REGION Network 20
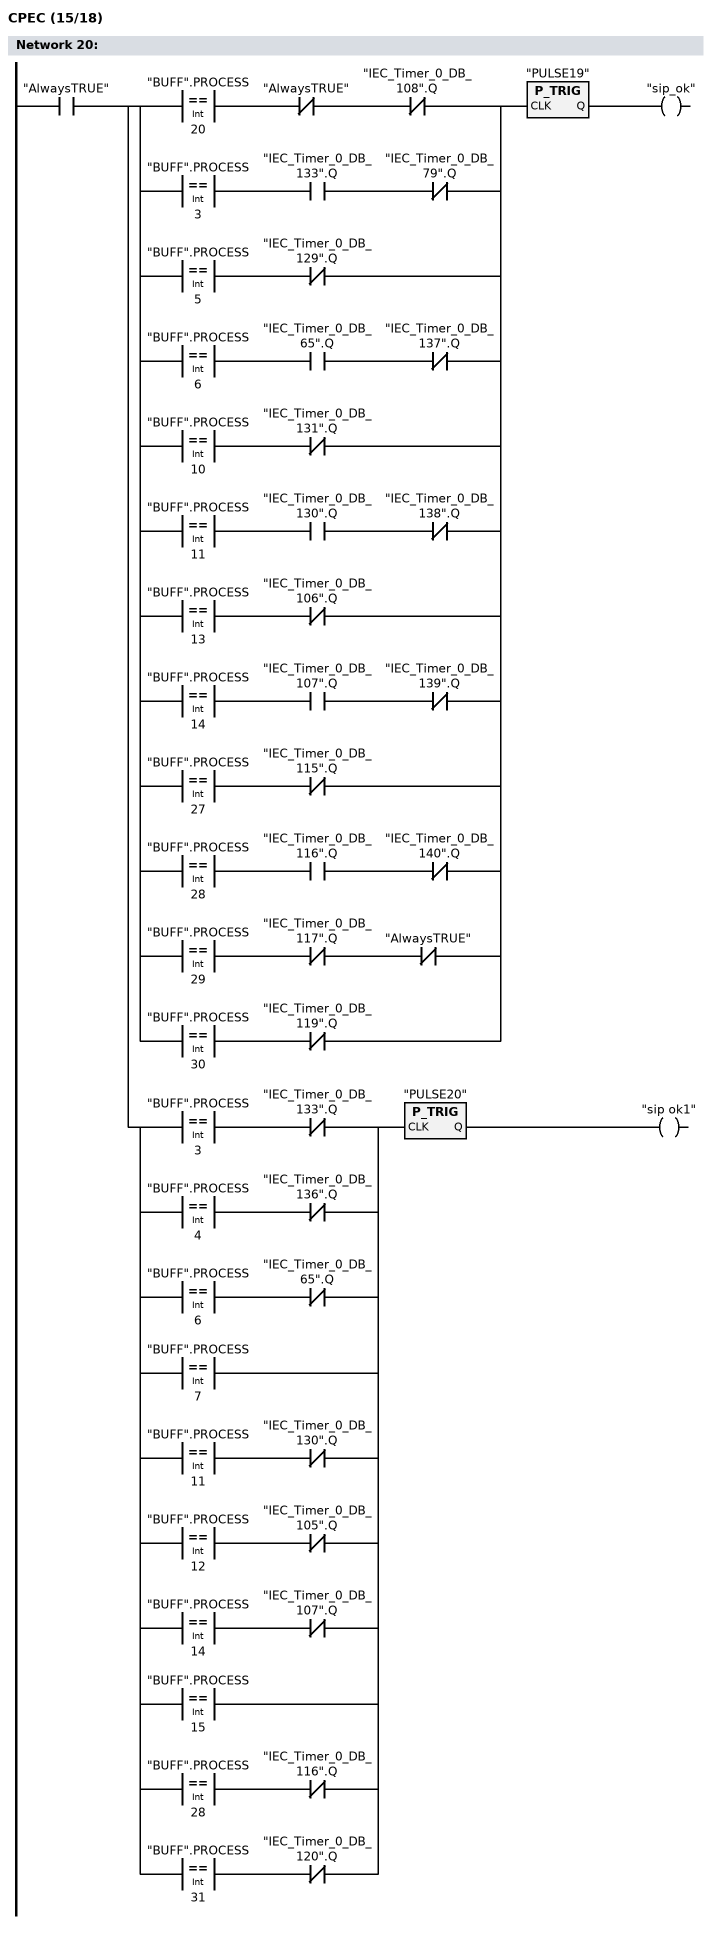
   RUNG wire#powerrail
      Contact( "AlwaysTRUE" )
      wire#w1
      { S7_Templates := "SrcType := Int" } EQ_Contact(in1 := "BUFF".PROCESS, in2 := 20)
      I_Contact( "AlwaysTRUE" )
      I_Contact( "IEC_Timer_0_DB_108".Q )
      wire#w2
      P_Trig( "PULSE19" )
      Coil( "sip_ok" )
   END_RUNG
   RUNG wire#w1
      { S7_Templates := "SrcType := Int" } EQ_Contact(in1 := "BUFF".PROCESS, in2 := 3)
      Contact( "IEC_Timer_0_DB_133".Q )
      I_Contact( "IEC_Timer_0_DB_79".Q )
   END_RUNG wire#w2
   RUNG wire#w1
      { S7_Templates := "SrcType := Int" } EQ_Contact(in1 := "BUFF".PROCESS, in2 := 5)
      I_Contact( "IEC_Timer_0_DB_129".Q )
   END_RUNG wire#w2
   RUNG wire#w1
      { S7_Templates := "SrcType := Int" } EQ_Contact(in1 := "BUFF".PROCESS, in2 := 6)
      Contact( "IEC_Timer_0_DB_65".Q )
      I_Contact( "IEC_Timer_0_DB_137".Q )
   END_RUNG wire#w2
   RUNG wire#w1
      { S7_Templates := "SrcType := Int" } EQ_Contact(in1 := "BUFF".PROCESS, in2 := 10)
      I_Contact( "IEC_Timer_0_DB_131".Q )
   END_RUNG wire#w2
   RUNG wire#w1
      { S7_Templates := "SrcType := Int" } EQ_Contact(in1 := "BUFF".PROCESS, in2 := 11)
      Contact( "IEC_Timer_0_DB_130".Q )
      I_Contact( "IEC_Timer_0_DB_138".Q )
   END_RUNG wire#w2
   RUNG wire#w1
      { S7_Templates := "SrcType := Int" } EQ_Contact(in1 := "BUFF".PROCESS, in2 := 13)
      I_Contact( "IEC_Timer_0_DB_106".Q )
   END_RUNG wire#w2
   RUNG wire#w1
      { S7_Templates := "SrcType := Int" } EQ_Contact(in1 := "BUFF".PROCESS, in2 := 14)
      Contact( "IEC_Timer_0_DB_107".Q )
      I_Contact( "IEC_Timer_0_DB_139".Q )
   END_RUNG wire#w2
   RUNG wire#w1
      { S7_Templates := "SrcType := Int" } EQ_Contact(in1 := "BUFF".PROCESS, in2 := 27)
      I_Contact( "IEC_Timer_0_DB_115".Q )
   END_RUNG wire#w2
   RUNG wire#w1
      { S7_Templates := "SrcType := Int" } EQ_Contact(in1 := "BUFF".PROCESS, in2 := 28)
      Contact( "IEC_Timer_0_DB_116".Q )
      I_Contact( "IEC_Timer_0_DB_140".Q )
   END_RUNG wire#w2
   RUNG wire#w1
      { S7_Templates := "SrcType := Int" } EQ_Contact(in1 := "BUFF".PROCESS, in2 := 29)
      I_Contact( "IEC_Timer_0_DB_117".Q )
      I_Contact( "AlwaysTRUE" )
   END_RUNG wire#w2
   RUNG wire#w1
      { S7_Templates := "SrcType := Int" } EQ_Contact(in1 := "BUFF".PROCESS, in2 := 30)
      I_Contact( "IEC_Timer_0_DB_119".Q )
   END_RUNG wire#w2
   RUNG wire#w1
      { S7_Templates := "SrcType := Int" } EQ_Contact(in1 := "BUFF".PROCESS, in2 := 3)
      I_Contact( "IEC_Timer_0_DB_133".Q )
      wire#w3
      P_Trig( "PULSE20" )
      Coil( "sip ok1" )
   END_RUNG
   RUNG wire#w1
      { S7_Templates := "SrcType := Int" } EQ_Contact(in1 := "BUFF".PROCESS, in2 := 4)
      I_Contact( "IEC_Timer_0_DB_136".Q )
   END_RUNG wire#w3
   RUNG wire#w1
      { S7_Templates := "SrcType := Int" } EQ_Contact(in1 := "BUFF".PROCESS, in2 := 6)
      I_Contact( "IEC_Timer_0_DB_65".Q )
   END_RUNG wire#w3
   RUNG wire#w1
      { S7_Templates := "SrcType := Int" } EQ_Contact(in1 := "BUFF".PROCESS, in2 := 7)
   END_RUNG wire#w3
   RUNG wire#w1
      { S7_Templates := "SrcType := Int" } EQ_Contact(in1 := "BUFF".PROCESS, in2 := 11)
      I_Contact( "IEC_Timer_0_DB_130".Q )
   END_RUNG wire#w3
   RUNG wire#w1
      { S7_Templates := "SrcType := Int" } EQ_Contact(in1 := "BUFF".PROCESS, in2 := 12)
      I_Contact( "IEC_Timer_0_DB_105".Q )
   END_RUNG wire#w3
   RUNG wire#w1
      { S7_Templates := "SrcType := Int" } EQ_Contact(in1 := "BUFF".PROCESS, in2 := 14)
      I_Contact( "IEC_Timer_0_DB_107".Q )
   END_RUNG wire#w3
   RUNG wire#w1
      { S7_Templates := "SrcType := Int" } EQ_Contact(in1 := "BUFF".PROCESS, in2 := 15)
   END_RUNG wire#w3
   RUNG wire#w1
      { S7_Templates := "SrcType := Int" } EQ_Contact(in1 := "BUFF".PROCESS, in2 := 28)
      I_Contact( "IEC_Timer_0_DB_116".Q )
   END_RUNG wire#w3
   RUNG wire#w1
      { S7_Templates := "SrcType := Int" } EQ_Contact(in1 := "BUFF".PROCESS, in2 := 31)
      I_Contact( "IEC_Timer_0_DB_120".Q )
   END_RUNG wire#w3
   // the same network as SCL:
   #_w1 := "AlwaysTRUE" AND ((("BUFF".PROCESS = 20) AND NOT "AlwaysTRUE" AND NOT "IEC_Timer_0_DB_108".Q) OR (("BUFF".PROCESS = 3) AND "IEC_Timer_0_DB_133".Q AND NOT "IEC_Timer_0_DB_79".Q) OR (("BUFF".PROCESS = 5) AND NOT "IEC_Timer_0_DB_129".Q) OR (("BUFF".PROCESS = 6) AND "IEC_Timer_0_DB_65".Q AND NOT "IEC_Timer_0_DB_137".Q) OR (("BUFF".PROCESS = 10) AND NOT "IEC_Timer_0_DB_131".Q) OR (("BUFF".PROCESS = 11) AND "IEC_Timer_0_DB_130".Q AND NOT "IEC_Timer_0_DB_138".Q) OR (("BUFF".PROCESS = 13) AND NOT "IEC_Timer_0_DB_106".Q) OR (("BUFF".PROCESS = 14) AND "IEC_Timer_0_DB_107".Q AND NOT "IEC_Timer_0_DB_139".Q) OR (("BUFF".PROCESS = 27) AND NOT "IEC_Timer_0_DB_115".Q) OR (("BUFF".PROCESS = 28) AND "IEC_Timer_0_DB_116".Q AND NOT "IEC_Timer_0_DB_140".Q) OR (("BUFF".PROCESS = 29) AND NOT "IEC_Timer_0_DB_117".Q AND NOT "AlwaysTRUE") OR (("BUFF".PROCESS = 30) AND NOT "IEC_Timer_0_DB_119".Q));
   #_w2 := #_w1 AND NOT "PULSE19";   // rising edge
   "PULSE19" := #_w1;
   "sip_ok" := #_w2;
   #_w3 := "AlwaysTRUE" AND ((("BUFF".PROCESS = 3) AND NOT "IEC_Timer_0_DB_133".Q) OR (("BUFF".PROCESS = 4) AND NOT "IEC_Timer_0_DB_136".Q) OR (("BUFF".PROCESS = 6) AND NOT "IEC_Timer_0_DB_65".Q) OR ("BUFF".PROCESS = 7) OR (("BUFF".PROCESS = 11) AND NOT "IEC_Timer_0_DB_130".Q) OR (("BUFF".PROCESS = 12) AND NOT "IEC_Timer_0_DB_105".Q) OR (("BUFF".PROCESS = 14) AND NOT "IEC_Timer_0_DB_107".Q) OR ("BUFF".PROCESS = 15) OR (("BUFF".PROCESS = 28) AND NOT "IEC_Timer_0_DB_116".Q) OR (("BUFF".PROCESS = 31) AND NOT "IEC_Timer_0_DB_120".Q));
   #_w4 := #_w3 AND NOT "PULSE20";   // rising edge
   "PULSE20" := #_w3;
   "sip ok1" := #_w4;
END_REGION

REGION Network 21
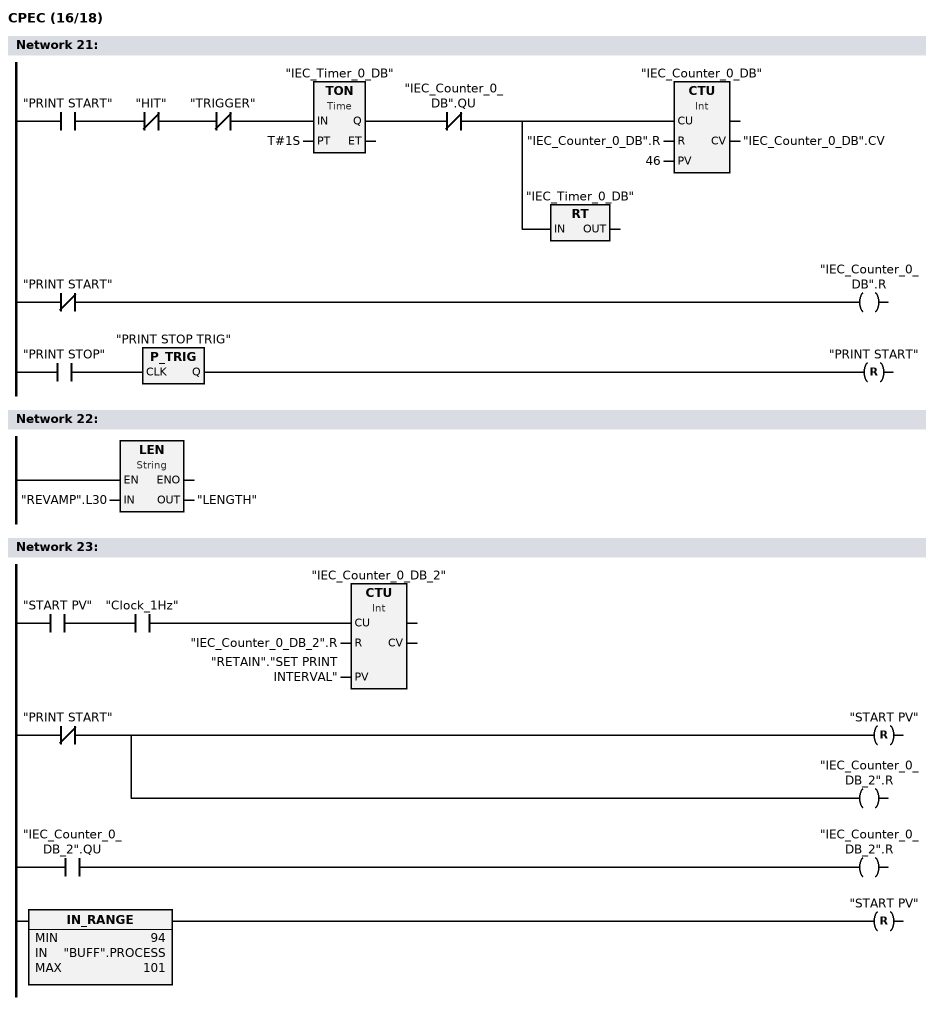
   RUNG wire#powerrail
      Contact( "PRINT START" )
      I_Contact( "HIT" )
      I_Contact( "TRIGGER" )
      { S7_Templates := "time_type := Time" } "IEC_Timer_0_DB".TON(pt := T#1S, et =>)
      I_Contact( "IEC_Counter_0_DB".QU )
      wire#w1
      { S7_Templates := "value_type := Int" } "IEC_Counter_0_DB".CTU(r := "IEC_Counter_0_DB".R, pv := 46, cv => "IEC_Counter_0_DB".CV)
   END_RUNG
   RUNG wire#w1
      RT_Coil( "IEC_Timer_0_DB" )
   END_RUNG
   RUNG wire#powerrail
      I_Contact( "PRINT START" )
      Coil( "IEC_Counter_0_DB".R )
   END_RUNG
   RUNG wire#powerrail
      Contact( "PRINT STOP" )
      P_Trig( "PRINT STOP TRIG" )
      R_Coil( "PRINT START" )
   END_RUNG
   // the same network as SCL:
   "IEC_Timer_0_DB".TON(IN := "PRINT START" AND NOT "HIT" AND NOT "TRIGGER", PT := T#1S);
   #_w1 := "IEC_Timer_0_DB".Q AND NOT "IEC_Counter_0_DB".QU;
   "IEC_Counter_0_DB".CTU(CU := #_w1, R := "IEC_Counter_0_DB".R, PV := 46, CV => "IEC_Counter_0_DB".CV);
   IF #_w1 THEN RESET_TIMER("IEC_Timer_0_DB"); END_IF;
   "IEC_Counter_0_DB".R := NOT "PRINT START";
   #_w2 := "PRINT STOP" AND NOT "PRINT STOP TRIG";   // rising edge
   "PRINT STOP TRIG" := "PRINT STOP";
   IF #_w2 THEN "PRINT START" := FALSE; END_IF;
END_REGION

REGION Network 22
   RUNG wire#powerrail
      { S7_Templates := "[str_type := String, return_type := Int]" } LEN(IN := "REVAMP".L30, OUT => "LENGTH")
   END_RUNG
   // the same network as SCL:
   LEN(IN := "REVAMP".L30, OUT => "LENGTH");
END_REGION

REGION Network 23
   RUNG wire#powerrail
      Contact( "START PV" )
      Contact( "Clock_1Hz" )
      { S7_Templates := "value_type := Int" } "IEC_Counter_0_DB_2".CTU(r := "IEC_Counter_0_DB_2".R, pv := "RETAIN"."SET PRINT INTERVAL", cv =>)
   END_RUNG
   RUNG wire#powerrail
      I_Contact( "PRINT START" )
      wire#w1
      R_Coil( "START PV" )
   END_RUNG
   RUNG wire#w1
      Coil( "IEC_Counter_0_DB_2".R )
   END_RUNG
   RUNG wire#powerrail
      Contact( "IEC_Counter_0_DB_2".QU )
      Coil( "IEC_Counter_0_DB_2".R )
   END_RUNG
   RUNG wire#powerrail
      { S7_Templates := "SrcType := Int" } InRange(min := 94, in := "BUFF".PROCESS, max := 101)
      R_Coil( "START PV" )
   END_RUNG
   // the same network as SCL:
   "IEC_Counter_0_DB_2".CTU(CU := "START PV" AND "Clock_1Hz",
                           R := "IEC_Counter_0_DB_2".R,
                           PV := "RETAIN"."SET PRINT INTERVAL");
   IF NOT "PRINT START" THEN "START PV" := FALSE; END_IF;
   "IEC_Counter_0_DB_2".R := NOT "PRINT START";
   "IEC_Counter_0_DB_2".R := "IEC_Counter_0_DB_2".QU;
   IF (94 <= "BUFF".PROCESS) AND ("BUFF".PROCESS <= 101) THEN "START PV" := FALSE; END_IF;
END_REGION

REGION Network 24
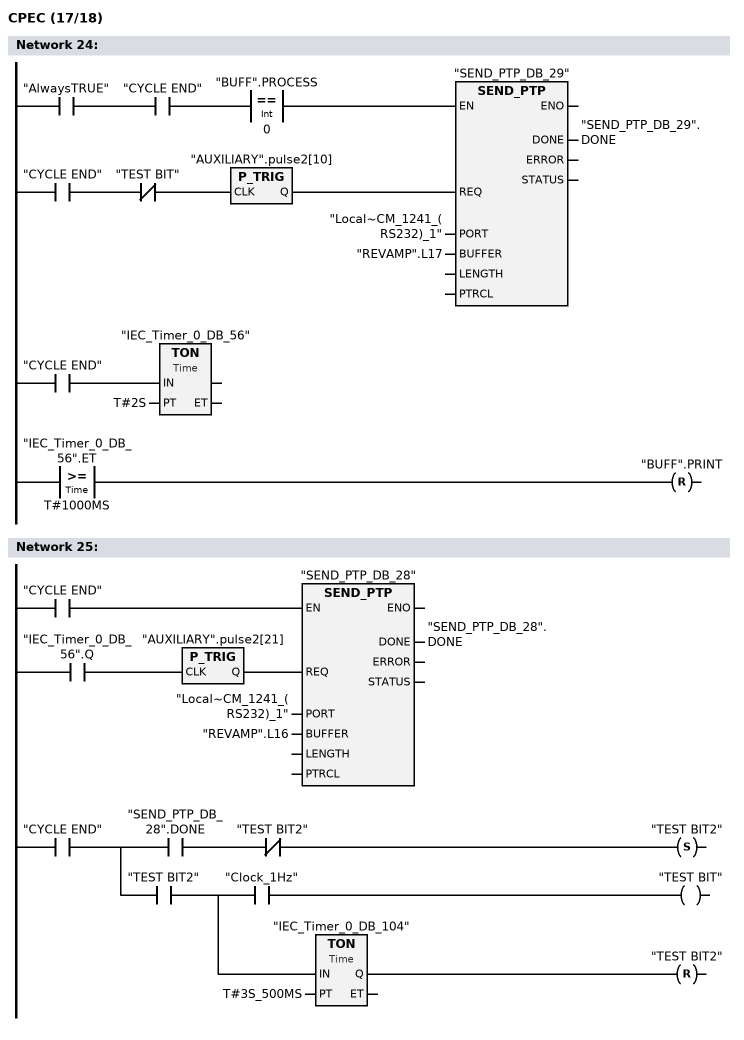
   RUNG wire#powerrail
      Contact( "AlwaysTRUE" )
      Contact( "CYCLE END" )
      { S7_Templates := "SrcType := Int" } EQ_Contact(in1 := "BUFF".PROCESS, in2 := 0)
      "SEND_PTP_DB_29".SEND_PTP(REQ := wire#w1, PORT := "Local~CM_1241_(RS232)_1", BUFFER := "REVAMP".L17, LENGTH :=, PTRCL :=, DONE => "SEND_PTP_DB_29".DONE, ERROR =>, STATUS =>)
   END_RUNG
   RUNG wire#powerrail
      Contact( "CYCLE END" )
      I_Contact( "TEST BIT" )
      P_Trig( "AUXILIARY".pulse2[10] )
   END_RUNG wire#w1
   RUNG wire#powerrail
      Contact( "CYCLE END" )
      { S7_Templates := "time_type := Time" } "IEC_Timer_0_DB_56".TON(pt := T#2S, et =>)
   END_RUNG
   RUNG wire#powerrail
      { S7_Templates := "SrcType := Time" } GE_Contact(in1 := "IEC_Timer_0_DB_56".ET, in2 := T#1000MS)
      R_Coil( "BUFF".PRINT )
   END_RUNG
   // the same network as SCL:
   #_w1 := "CYCLE END" AND NOT "TEST BIT";
   #_w2 := #_w1 AND NOT "AUXILIARY".pulse2[10];   // rising edge
   "AUXILIARY".pulse2[10] := #_w1;
   IF "AlwaysTRUE" AND "CYCLE END" AND ("BUFF".PROCESS = 0) THEN
       "SEND_PTP_DB_29"(REQ := #_w2,   // SEND_PTP
                        PORT := "Local~CM_1241_(RS232)_1",
                        BUFFER := "REVAMP".L17,
                        DONE => "SEND_PTP_DB_29".DONE);
   END_IF;
   "IEC_Timer_0_DB_56".TON(IN := "CYCLE END", PT := T#2S);
   IF "IEC_Timer_0_DB_56".ET >= T#1000MS THEN "BUFF".PRINT := FALSE; END_IF;
END_REGION

REGION Network 25
   RUNG wire#powerrail
      Contact( "CYCLE END" )
      "SEND_PTP_DB_28".SEND_PTP(REQ := wire#w1, PORT := "Local~CM_1241_(RS232)_1", BUFFER := "REVAMP".L16, LENGTH :=, PTRCL :=, DONE => "SEND_PTP_DB_28".DONE, ERROR =>, STATUS =>)
   END_RUNG
   RUNG wire#powerrail
      Contact( "IEC_Timer_0_DB_56".Q )
      P_Trig( "AUXILIARY".pulse2[21] )
   END_RUNG wire#w1
   RUNG wire#powerrail
      Contact( "CYCLE END" )
      wire#w2
      Contact( "SEND_PTP_DB_28".DONE )
      I_Contact( "TEST BIT2" )
      S_Coil( "TEST BIT2" )
   END_RUNG
   RUNG wire#w2
      Contact( "TEST BIT2" )
      wire#w3
      Contact( "Clock_1Hz" )
      Coil( "TEST BIT" )
   END_RUNG
   RUNG wire#w3
      { S7_Templates := "time_type := Time" } "IEC_Timer_0_DB_104".TON(pt := T#3S_500MS, et =>)
      R_Coil( "TEST BIT2" )
   END_RUNG
   // the same network as SCL:
   #_w1 := "IEC_Timer_0_DB_56".Q AND NOT "AUXILIARY".pulse2[21];   // rising edge
   "AUXILIARY".pulse2[21] := "IEC_Timer_0_DB_56".Q;
   IF "CYCLE END" THEN
       "SEND_PTP_DB_28"(REQ := #_w1,   // SEND_PTP
                        PORT := "Local~CM_1241_(RS232)_1",
                        BUFFER := "REVAMP".L16,
                        DONE => "SEND_PTP_DB_28".DONE);
   END_IF;
   IF "CYCLE END" AND "SEND_PTP_DB_28".DONE AND NOT "TEST BIT2" THEN "TEST BIT2" := TRUE; END_IF;
   #_w2 := "CYCLE END" AND "TEST BIT2";
   "TEST BIT" := #_w2 AND "Clock_1Hz";
   "IEC_Timer_0_DB_104".TON(IN := #_w2, PT := T#3S_500MS);
   IF "IEC_Timer_0_DB_104".Q THEN "TEST BIT2" := FALSE; END_IF;
END_REGION

REGION Network 26
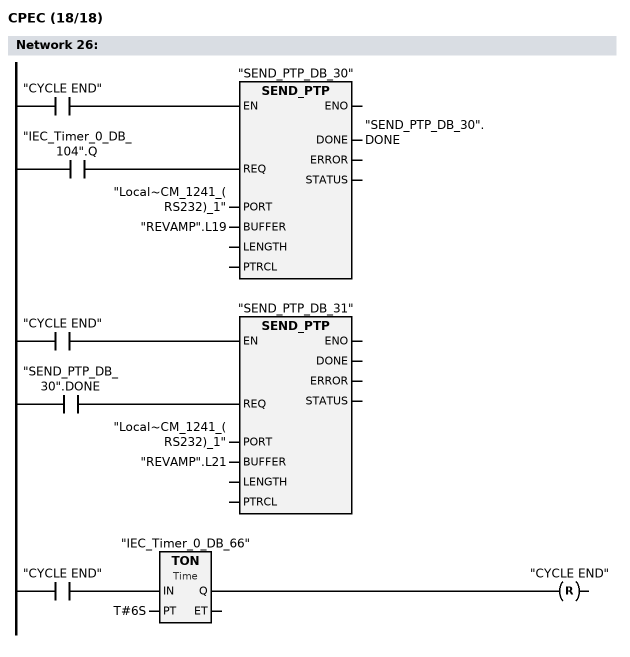
   RUNG wire#powerrail
      Contact( "CYCLE END" )
      "SEND_PTP_DB_30".SEND_PTP(REQ := wire#w1, PORT := "Local~CM_1241_(RS232)_1", BUFFER := "REVAMP".L19, LENGTH :=, PTRCL :=, DONE => "SEND_PTP_DB_30".DONE, ERROR =>, STATUS =>)
   END_RUNG
   RUNG wire#powerrail
      Contact( "IEC_Timer_0_DB_104".Q )
   END_RUNG wire#w1
   RUNG wire#powerrail
      Contact( "CYCLE END" )
      "SEND_PTP_DB_31".SEND_PTP(REQ := wire#w2, PORT := "Local~CM_1241_(RS232)_1", BUFFER := "REVAMP".L21, LENGTH :=, PTRCL :=, DONE =>, ERROR =>, STATUS =>)
   END_RUNG
   RUNG wire#powerrail
      Contact( "SEND_PTP_DB_30".DONE )
   END_RUNG wire#w2
   RUNG wire#powerrail
      Contact( "CYCLE END" )
      { S7_Templates := "time_type := Time" } "IEC_Timer_0_DB_66".TON(pt := T#6S, et =>)
      R_Coil( "CYCLE END" )
   END_RUNG
   // the same network as SCL:
   IF "CYCLE END" THEN
       "SEND_PTP_DB_30"(REQ := "IEC_Timer_0_DB_104".Q,   // SEND_PTP
                        PORT := "Local~CM_1241_(RS232)_1",
                        BUFFER := "REVAMP".L19,
                        DONE => "SEND_PTP_DB_30".DONE);
   END_IF;
   IF "CYCLE END" THEN
       "SEND_PTP_DB_31"(REQ := "SEND_PTP_DB_30".DONE, PORT := "Local~CM_1241_(RS232)_1", BUFFER := "REVAMP".L21);   // SEND_PTP
   END_IF;
   "IEC_Timer_0_DB_66".TON(IN := "CYCLE END", PT := T#6S);
   IF "IEC_Timer_0_DB_66".Q THEN "CYCLE END" := FALSE; END_IF;
END_REGION
END_FUNCTION
